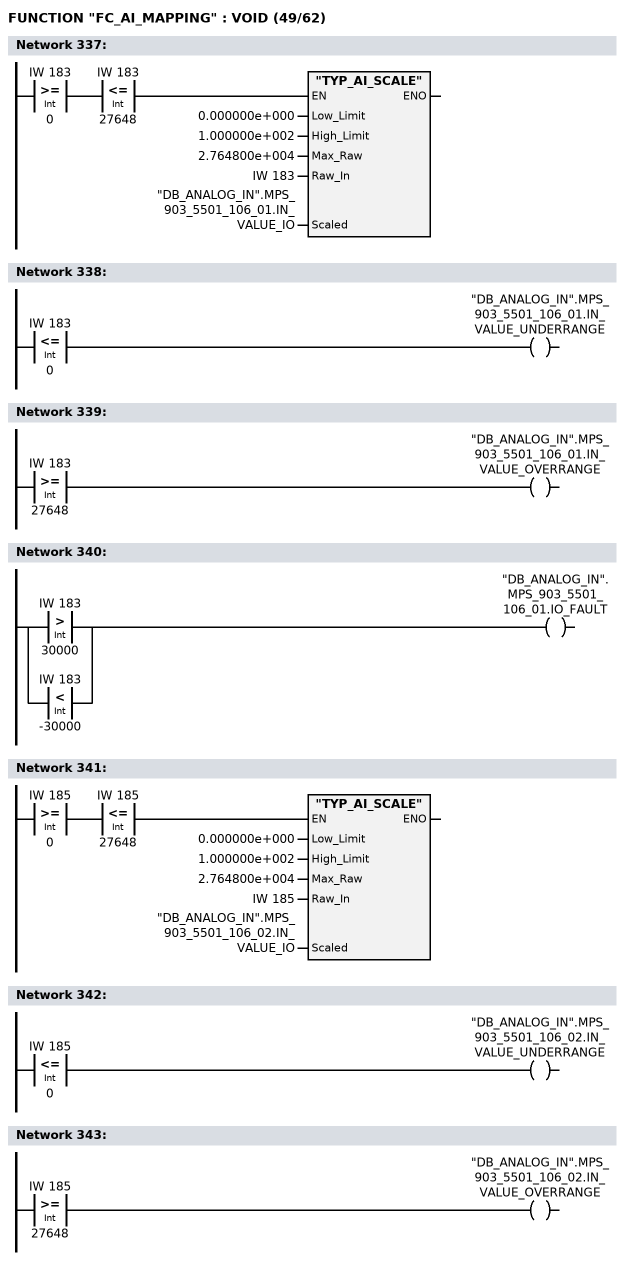

      A(    ;
      L     IW      183;
      L     0;
      >=I   ;
      )     ;
      A(    ;
      L     IW      183;

      L     27648;
      <=I   ;
      )     ;
      JNB   _055;
      CALL "TYP_AI_SCALE" (
           Low_Limit                := 0.000000e+000,
           High_Limit               := 1.000000e+002,
           Max_Raw                  := 2.764800e+004,
           Raw_In                   := IW      183,
           Scaled                   := "DB_ANALOG_IN".MPS_903_5501_106_01.IN_VALUE_IO);
_055: NOP   0;
NETWORK
TITLE =

      L     IW      183;
      L     0;
      <=I   ;
      =     "DB_ANALOG_IN".MPS_903_5501_106_01.IN_VALUE_UNDERRANGE;
NETWORK
TITLE =

      L     IW      183;
      L     27648;
      >=I   ;
      =     "DB_ANALOG_IN".MPS_903_5501_106_01.IN_VALUE_OVERRANGE;
NETWORK
TITLE =

      O(    ;
      L     IW      183;
      L     30000;
      >I    ;
      )     ;
      O(    ;
      L     IW      183;
      L     -30000;
      <I    ;
      )     ;
      =     "DB_ANALOG_IN".MPS_903_5501_106_01.IO_FAULT;

NETWORK
TITLE =

      A(    ;
      L     IW      185;
      L     0;
      >=I   ;
      )     ;
      A(    ;
      L     IW      185;

      L     27648;
      <=I   ;
      )     ;
      JNB   _056;
      CALL "TYP_AI_SCALE" (
           Low_Limit                := 0.000000e+000,
           High_Limit               := 1.000000e+002,
           Max_Raw                  := 2.764800e+004,
           Raw_In                   := IW      185,
           Scaled                   := "DB_ANALOG_IN".MPS_903_5501_106_02.IN_VALUE_IO);
_056: NOP   0;
NETWORK
TITLE =

      L     IW      185;
      L     0;
      <=I   ;
      =     "DB_ANALOG_IN".MPS_903_5501_106_02.IN_VALUE_UNDERRANGE;
NETWORK
TITLE =

      L     IW      185;
      L     27648;
      >=I   ;
      =     "DB_ANALOG_IN".MPS_903_5501_106_02.IN_VALUE_OVERRANGE;
NETWORK
TITLE =
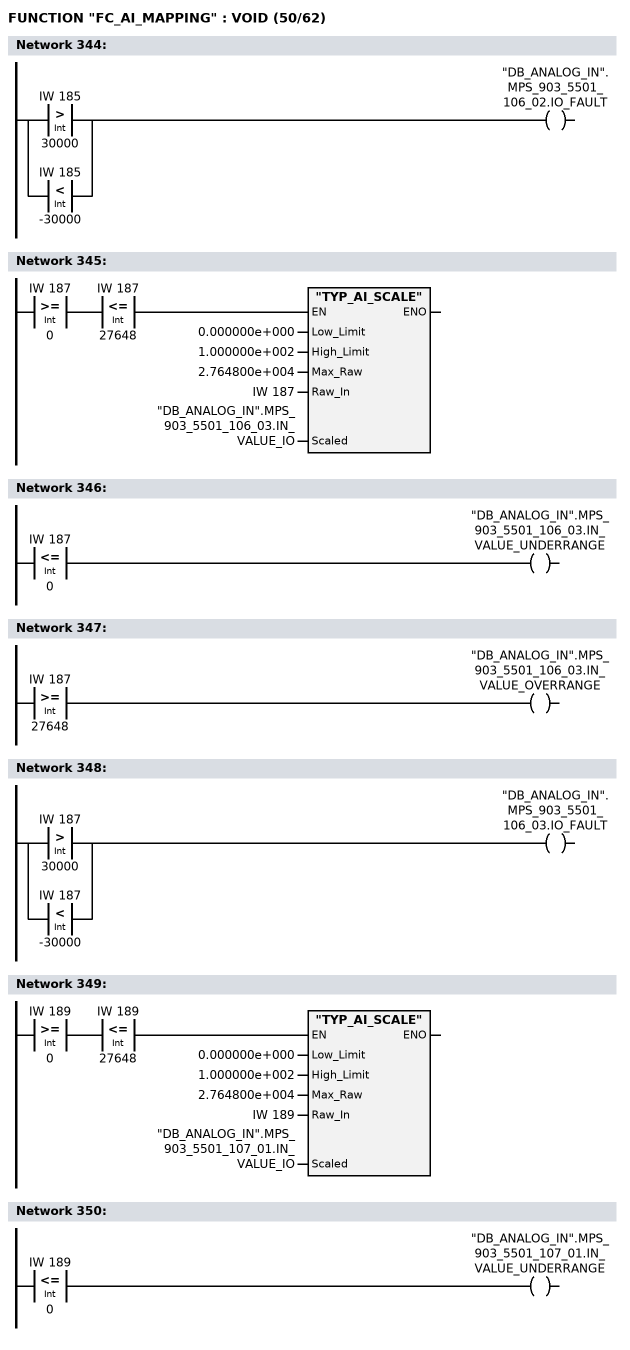

      O(    ;
      L     IW      185;
      L     30000;
      >I    ;
      )     ;
      O(    ;
      L     IW      185;
      L     -30000;
      <I    ;
      )     ;
      =     "DB_ANALOG_IN".MPS_903_5501_106_02.IO_FAULT;

NETWORK
TITLE =

      A(    ;
      L     IW      187;
      L     0;
      >=I   ;
      )     ;
      A(    ;
      L     IW      187;

      L     27648;
      <=I   ;
      )     ;
      JNB   _057;
      CALL "TYP_AI_SCALE" (
           Low_Limit                := 0.000000e+000,
           High_Limit               := 1.000000e+002,
           Max_Raw                  := 2.764800e+004,
           Raw_In                   := IW      187,
           Scaled                   := "DB_ANALOG_IN".MPS_903_5501_106_03.IN_VALUE_IO);
_057: NOP   0;
NETWORK
TITLE =

      L     IW      187;
      L     0;
      <=I   ;
      =     "DB_ANALOG_IN".MPS_903_5501_106_03.IN_VALUE_UNDERRANGE;
NETWORK
TITLE =

      L     IW      187;
      L     27648;
      >=I   ;
      =     "DB_ANALOG_IN".MPS_903_5501_106_03.IN_VALUE_OVERRANGE;
NETWORK
TITLE =

      O(    ;
      L     IW      187;
      L     30000;
      >I    ;
      )     ;
      O(    ;
      L     IW      187;
      L     -30000;
      <I    ;
      )     ;
      =     "DB_ANALOG_IN".MPS_903_5501_106_03.IO_FAULT;

NETWORK
TITLE =

      A(    ;
      L     IW      189;
      L     0;
      >=I   ;
      )     ;
      A(    ;
      L     IW      189;

      L     27648;
      <=I   ;
      )     ;
      JNB   _058;
      CALL "TYP_AI_SCALE" (
           Low_Limit                := 0.000000e+000,
           High_Limit               := 1.000000e+002,
           Max_Raw                  := 2.764800e+004,
           Raw_In                   := IW      189,
           Scaled                   := "DB_ANALOG_IN".MPS_903_5501_107_01.IN_VALUE_IO);
_058: NOP   0;
NETWORK
TITLE =

      L     IW      189;
      L     0;
      <=I   ;
      =     "DB_ANALOG_IN".MPS_903_5501_107_01.IN_VALUE_UNDERRANGE;
NETWORK
TITLE =
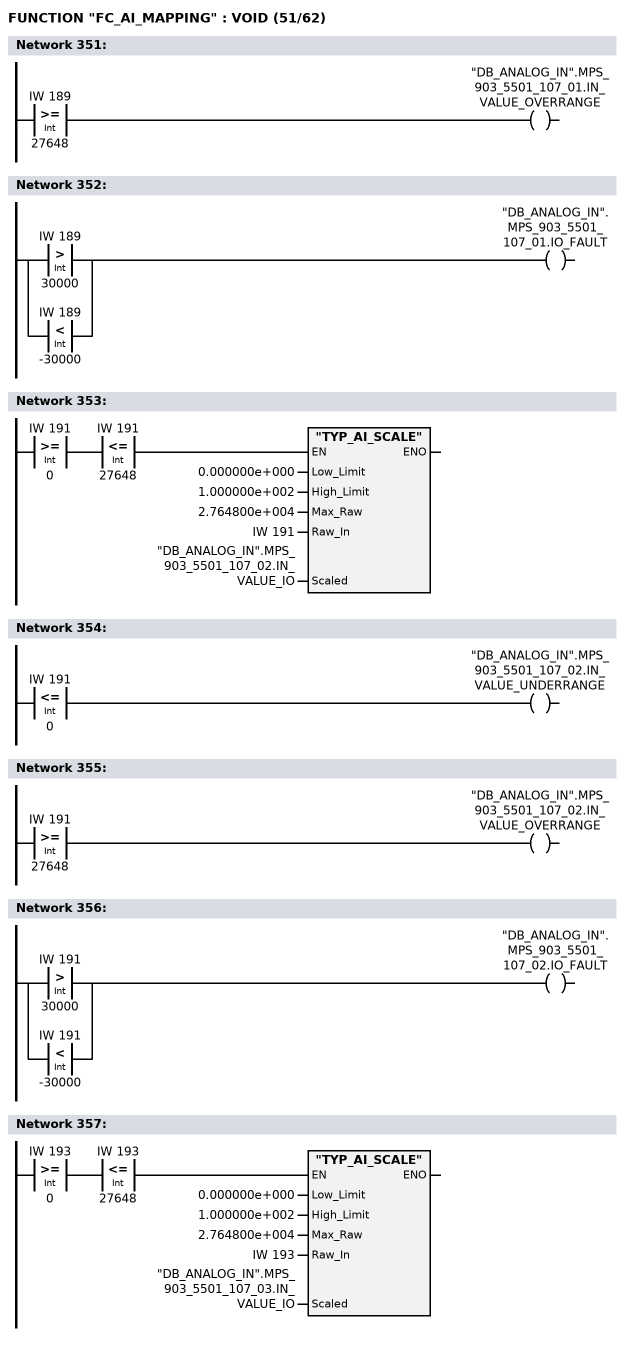

      L     IW      189;
      L     27648;
      >=I   ;
      =     "DB_ANALOG_IN".MPS_903_5501_107_01.IN_VALUE_OVERRANGE;
NETWORK
TITLE =

      O(    ;
      L     IW      189;
      L     30000;
      >I    ;
      )     ;
      O(    ;
      L     IW      189;
      L     -30000;
      <I    ;
      )     ;
      =     "DB_ANALOG_IN".MPS_903_5501_107_01.IO_FAULT;

NETWORK
TITLE =

      A(    ;
      L     IW      191;
      L     0;
      >=I   ;
      )     ;
      A(    ;
      L     IW      191;

      L     27648;
      <=I   ;
      )     ;
      JNB   _059;
      CALL "TYP_AI_SCALE" (
           Low_Limit                := 0.000000e+000,
           High_Limit               := 1.000000e+002,
           Max_Raw                  := 2.764800e+004,
           Raw_In                   := IW      191,
           Scaled                   := "DB_ANALOG_IN".MPS_903_5501_107_02.IN_VALUE_IO);
_059: NOP   0;
NETWORK
TITLE =

      L     IW      191;
      L     0;
      <=I   ;
      =     "DB_ANALOG_IN".MPS_903_5501_107_02.IN_VALUE_UNDERRANGE;
NETWORK
TITLE =

      L     IW      191;
      L     27648;
      >=I   ;
      =     "DB_ANALOG_IN".MPS_903_5501_107_02.IN_VALUE_OVERRANGE;
NETWORK
TITLE =

      O(    ;
      L     IW      191;
      L     30000;
      >I    ;
      )     ;
      O(    ;
      L     IW      191;
      L     -30000;
      <I    ;
      )     ;
      =     "DB_ANALOG_IN".MPS_903_5501_107_02.IO_FAULT;

NETWORK
TITLE =

      A(    ;
      L     IW      193;
      L     0;
      >=I   ;
      )     ;
      A(    ;
      L     IW      193;

      L     27648;
      <=I   ;
      )     ;
      JNB   _05a;
      CALL "TYP_AI_SCALE" (
           Low_Limit                := 0.000000e+000,
           High_Limit               := 1.000000e+002,
           Max_Raw                  := 2.764800e+004,
           Raw_In                   := IW      193,
           Scaled                   := "DB_ANALOG_IN".MPS_903_5501_107_03.IN_VALUE_IO);
_05a: NOP   0;
NETWORK
TITLE =
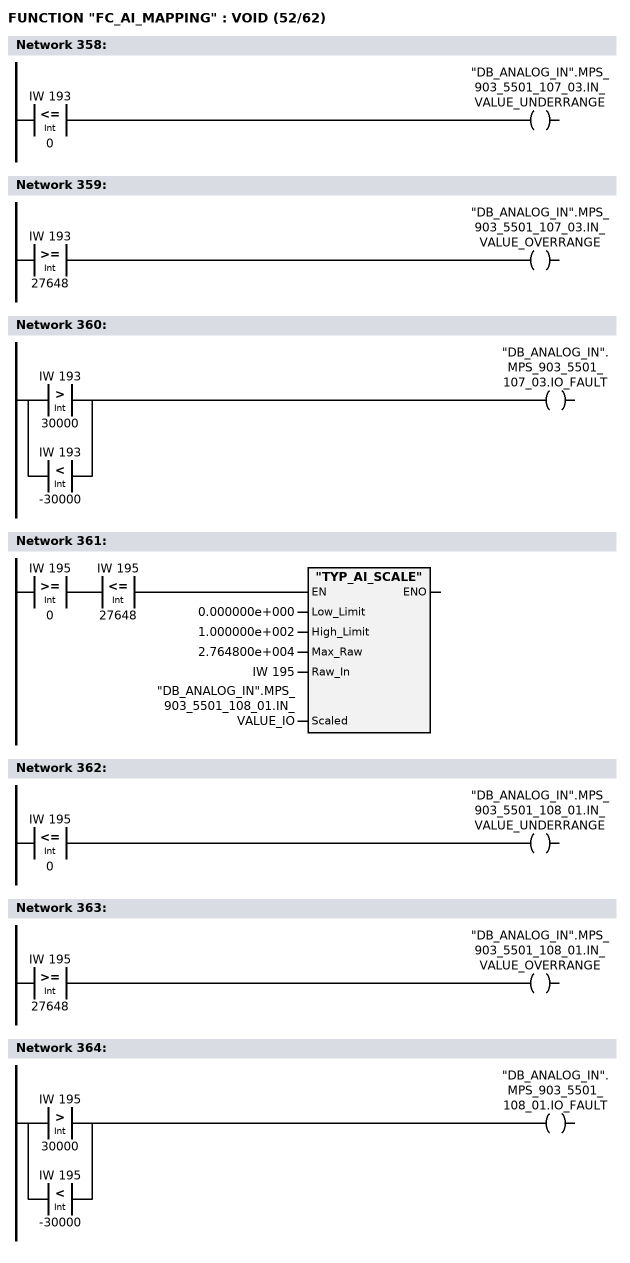

      L     IW      193;
      L     0;
      <=I   ;
      =     "DB_ANALOG_IN".MPS_903_5501_107_03.IN_VALUE_UNDERRANGE;
NETWORK
TITLE =

      L     IW      193;
      L     27648;
      >=I   ;
      =     "DB_ANALOG_IN".MPS_903_5501_107_03.IN_VALUE_OVERRANGE;
NETWORK
TITLE =

      O(    ;
      L     IW      193;
      L     30000;
      >I    ;
      )     ;
      O(    ;
      L     IW      193;
      L     -30000;
      <I    ;
      )     ;
      =     "DB_ANALOG_IN".MPS_903_5501_107_03.IO_FAULT;

NETWORK
TITLE =

      A(    ;
      L     IW      195;
      L     0;
      >=I   ;
      )     ;
      A(    ;
      L     IW      195;

      L     27648;
      <=I   ;
      )     ;
      JNB   _05b;
      CALL "TYP_AI_SCALE" (
           Low_Limit                := 0.000000e+000,
           High_Limit               := 1.000000e+002,
           Max_Raw                  := 2.764800e+004,
           Raw_In                   := IW      195,
           Scaled                   := "DB_ANALOG_IN".MPS_903_5501_108_01.IN_VALUE_IO);
_05b: NOP   0;
NETWORK
TITLE =

      L     IW      195;
      L     0;
      <=I   ;
      =     "DB_ANALOG_IN".MPS_903_5501_108_01.IN_VALUE_UNDERRANGE;
NETWORK
TITLE =

      L     IW      195;
      L     27648;
      >=I   ;
      =     "DB_ANALOG_IN".MPS_903_5501_108_01.IN_VALUE_OVERRANGE;
NETWORK
TITLE =

      O(    ;
      L     IW      195;
      L     30000;
      >I    ;
      )     ;
      O(    ;
      L     IW      195;
      L     -30000;
      <I    ;
      )     ;
      =     "DB_ANALOG_IN".MPS_903_5501_108_01.IO_FAULT;

NETWORK
TITLE =
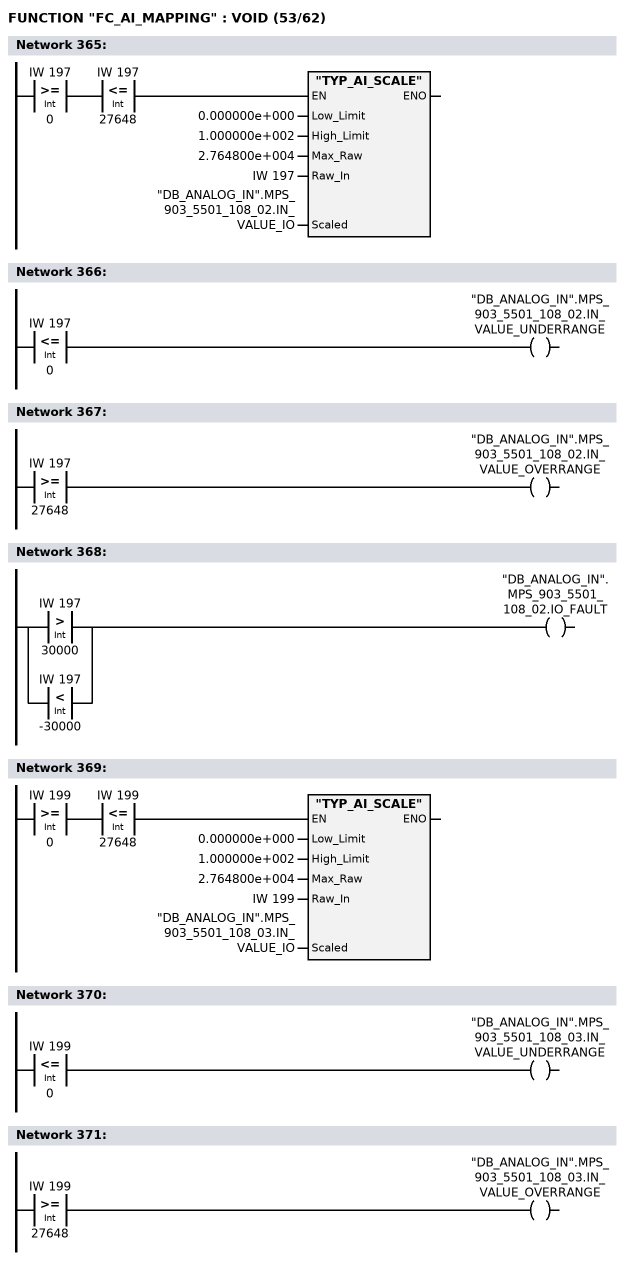

      A(    ;
      L     IW      197;
      L     0;
      >=I   ;
      )     ;
      A(    ;
      L     IW      197;

      L     27648;
      <=I   ;
      )     ;
      JNB   _05c;
      CALL "TYP_AI_SCALE" (
           Low_Limit                := 0.000000e+000,
           High_Limit               := 1.000000e+002,
           Max_Raw                  := 2.764800e+004,
           Raw_In                   := IW      197,
           Scaled                   := "DB_ANALOG_IN".MPS_903_5501_108_02.IN_VALUE_IO);
_05c: NOP   0;
NETWORK
TITLE =

      L     IW      197;
      L     0;
      <=I   ;
      =     "DB_ANALOG_IN".MPS_903_5501_108_02.IN_VALUE_UNDERRANGE;
NETWORK
TITLE =

      L     IW      197;
      L     27648;
      >=I   ;
      =     "DB_ANALOG_IN".MPS_903_5501_108_02.IN_VALUE_OVERRANGE;
NETWORK
TITLE =

      O(    ;
      L     IW      197;
      L     30000;
      >I    ;
      )     ;
      O(    ;
      L     IW      197;
      L     -30000;
      <I    ;
      )     ;
      =     "DB_ANALOG_IN".MPS_903_5501_108_02.IO_FAULT;

NETWORK
TITLE =

      A(    ;
      L     IW      199;
      L     0;
      >=I   ;
      )     ;
      A(    ;
      L     IW      199;

      L     27648;
      <=I   ;
      )     ;
      JNB   _05d;
      CALL "TYP_AI_SCALE" (
           Low_Limit                := 0.000000e+000,
           High_Limit               := 1.000000e+002,
           Max_Raw                  := 2.764800e+004,
           Raw_In                   := IW      199,
           Scaled                   := "DB_ANALOG_IN".MPS_903_5501_108_03.IN_VALUE_IO);
_05d: NOP   0;
NETWORK
TITLE =

      L     IW      199;
      L     0;
      <=I   ;
      =     "DB_ANALOG_IN".MPS_903_5501_108_03.IN_VALUE_UNDERRANGE;
NETWORK
TITLE =

      L     IW      199;
      L     27648;
      >=I   ;
      =     "DB_ANALOG_IN".MPS_903_5501_108_03.IN_VALUE_OVERRANGE;
NETWORK
TITLE =
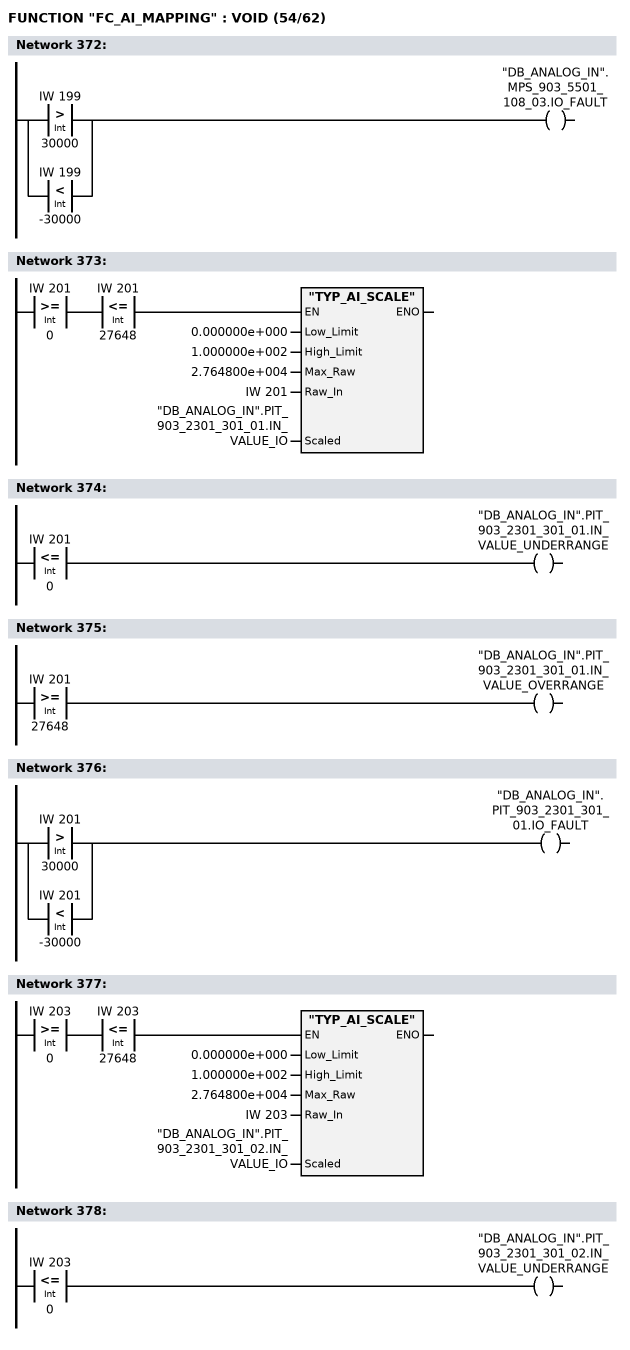

      O(    ;
      L     IW      199;
      L     30000;
      >I    ;
      )     ;
      O(    ;
      L     IW      199;
      L     -30000;
      <I    ;
      )     ;
      =     "DB_ANALOG_IN".MPS_903_5501_108_03.IO_FAULT;

NETWORK
TITLE =

      A(    ;
      L     IW      201;
      L     0;
      >=I   ;
      )     ;
      A(    ;
      L     IW      201;

      L     27648;
      <=I   ;
      )     ;
      JNB   _05e;
      CALL "TYP_AI_SCALE" (
           Low_Limit                := 0.000000e+000,
           High_Limit               := 1.000000e+002,
           Max_Raw                  := 2.764800e+004,
           Raw_In                   := IW      201,
           Scaled                   := "DB_ANALOG_IN".PIT_903_2301_301_01.IN_VALUE_IO);
_05e: NOP   0;
NETWORK
TITLE =

      L     IW      201;
      L     0;
      <=I   ;
      =     "DB_ANALOG_IN".PIT_903_2301_301_01.IN_VALUE_UNDERRANGE;
NETWORK
TITLE =

      L     IW      201;
      L     27648;
      >=I   ;
      =     "DB_ANALOG_IN".PIT_903_2301_301_01.IN_VALUE_OVERRANGE;
NETWORK
TITLE =

      O(    ;
      L     IW      201;
      L     30000;
      >I    ;
      )     ;
      O(    ;
      L     IW      201;
      L     -30000;
      <I    ;
      )     ;
      =     "DB_ANALOG_IN".PIT_903_2301_301_01.IO_FAULT;

NETWORK
TITLE =

      A(    ;
      L     IW      203;
      L     0;
      >=I   ;
      )     ;
      A(    ;
      L     IW      203;

      L     27648;
      <=I   ;
      )     ;
      JNB   _05f;
      CALL "TYP_AI_SCALE" (
           Low_Limit                := 0.000000e+000,
           High_Limit               := 1.000000e+002,
           Max_Raw                  := 2.764800e+004,
           Raw_In                   := IW      203,
           Scaled                   := "DB_ANALOG_IN".PIT_903_2301_301_02.IN_VALUE_IO);
_05f: NOP   0;
NETWORK
TITLE =

      L     IW      203;
      L     0;
      <=I   ;
      =     "DB_ANALOG_IN".PIT_903_2301_301_02.IN_VALUE_UNDERRANGE;
NETWORK
TITLE =
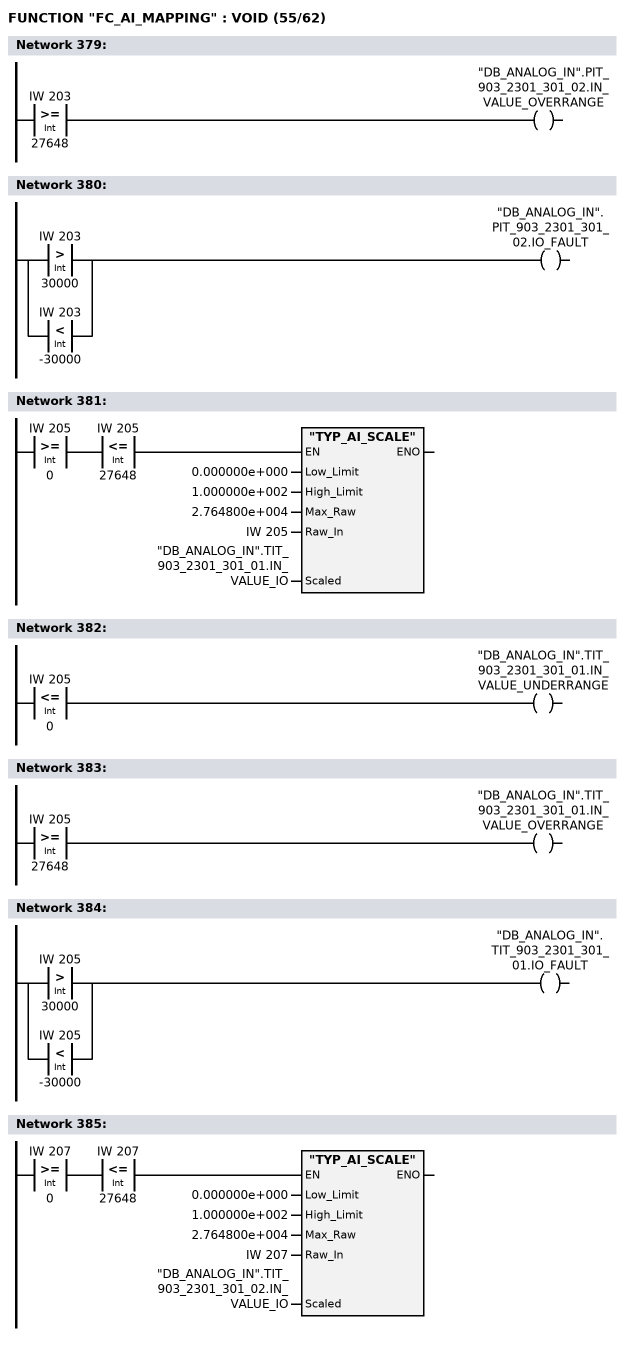

      L     IW      203;
      L     27648;
      >=I   ;
      =     "DB_ANALOG_IN".PIT_903_2301_301_02.IN_VALUE_OVERRANGE;
NETWORK
TITLE =

      O(    ;
      L     IW      203;
      L     30000;
      >I    ;
      )     ;
      O(    ;
      L     IW      203;
      L     -30000;
      <I    ;
      )     ;
      =     "DB_ANALOG_IN".PIT_903_2301_301_02.IO_FAULT;

NETWORK
TITLE =

      A(    ;
      L     IW      205;
      L     0;
      >=I   ;
      )     ;
      A(    ;
      L     IW      205;

      L     27648;
      <=I   ;
      )     ;
      JNB   _060;
      CALL "TYP_AI_SCALE" (
           Low_Limit                := 0.000000e+000,
           High_Limit               := 1.000000e+002,
           Max_Raw                  := 2.764800e+004,
           Raw_In                   := IW      205,
           Scaled                   := "DB_ANALOG_IN".TIT_903_2301_301_01.IN_VALUE_IO);
_060: NOP   0;
NETWORK
TITLE =

      L     IW      205;
      L     0;
      <=I   ;
      =     "DB_ANALOG_IN".TIT_903_2301_301_01.IN_VALUE_UNDERRANGE;
NETWORK
TITLE =

      L     IW      205;
      L     27648;
      >=I   ;
      =     "DB_ANALOG_IN".TIT_903_2301_301_01.IN_VALUE_OVERRANGE;
NETWORK
TITLE =

      O(    ;
      L     IW      205;
      L     30000;
      >I    ;
      )     ;
      O(    ;
      L     IW      205;
      L     -30000;
      <I    ;
      )     ;
      =     "DB_ANALOG_IN".TIT_903_2301_301_01.IO_FAULT;

NETWORK
TITLE =

      A(    ;
      L     IW      207;
      L     0;
      >=I   ;
      )     ;
      A(    ;
      L     IW      207;

      L     27648;
      <=I   ;
      )     ;
      JNB   _061;
      CALL "TYP_AI_SCALE" (
           Low_Limit                := 0.000000e+000,
           High_Limit               := 1.000000e+002,
           Max_Raw                  := 2.764800e+004,
           Raw_In                   := IW      207,
           Scaled                   := "DB_ANALOG_IN".TIT_903_2301_301_02.IN_VALUE_IO);
_061: NOP   0;
NETWORK
TITLE =
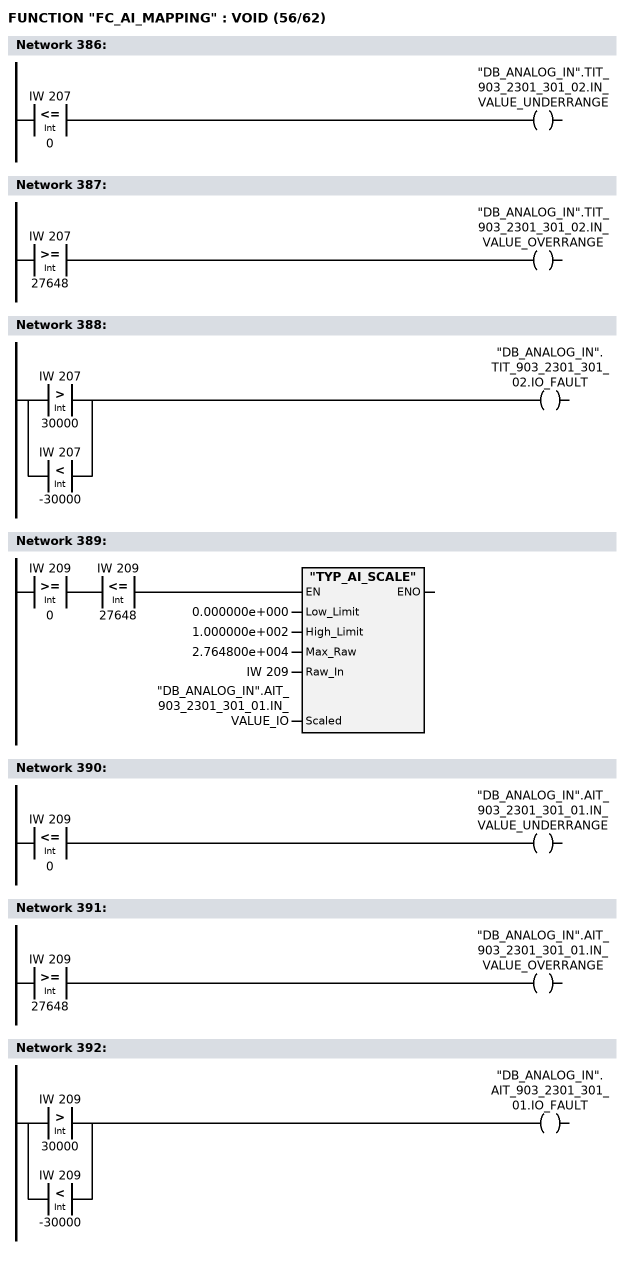

      L     IW      207;
      L     0;
      <=I   ;
      =     "DB_ANALOG_IN".TIT_903_2301_301_02.IN_VALUE_UNDERRANGE;
NETWORK
TITLE =

      L     IW      207;
      L     27648;
      >=I   ;
      =     "DB_ANALOG_IN".TIT_903_2301_301_02.IN_VALUE_OVERRANGE;
NETWORK
TITLE =

      O(    ;
      L     IW      207;
      L     30000;
      >I    ;
      )     ;
      O(    ;
      L     IW      207;
      L     -30000;
      <I    ;
      )     ;
      =     "DB_ANALOG_IN".TIT_903_2301_301_02.IO_FAULT;

NETWORK
TITLE =

      A(    ;
      L     IW      209;
      L     0;
      >=I   ;
      )     ;
      A(    ;
      L     IW      209;

      L     27648;
      <=I   ;
      )     ;
      JNB   _062;
      CALL "TYP_AI_SCALE" (
           Low_Limit                := 0.000000e+000,
           High_Limit               := 1.000000e+002,
           Max_Raw                  := 2.764800e+004,
           Raw_In                   := IW      209,
           Scaled                   := "DB_ANALOG_IN".AIT_903_2301_301_01.IN_VALUE_IO);
_062: NOP   0;
NETWORK
TITLE =

      L     IW      209;
      L     0;
      <=I   ;
      =     "DB_ANALOG_IN".AIT_903_2301_301_01.IN_VALUE_UNDERRANGE;
NETWORK
TITLE =

      L     IW      209;
      L     27648;
      >=I   ;
      =     "DB_ANALOG_IN".AIT_903_2301_301_01.IN_VALUE_OVERRANGE;
NETWORK
TITLE =

      O(    ;
      L     IW      209;
      L     30000;
      >I    ;
      )     ;
      O(    ;
      L     IW      209;
      L     -30000;
      <I    ;
      )     ;
      =     "DB_ANALOG_IN".AIT_903_2301_301_01.IO_FAULT;

NETWORK
TITLE =
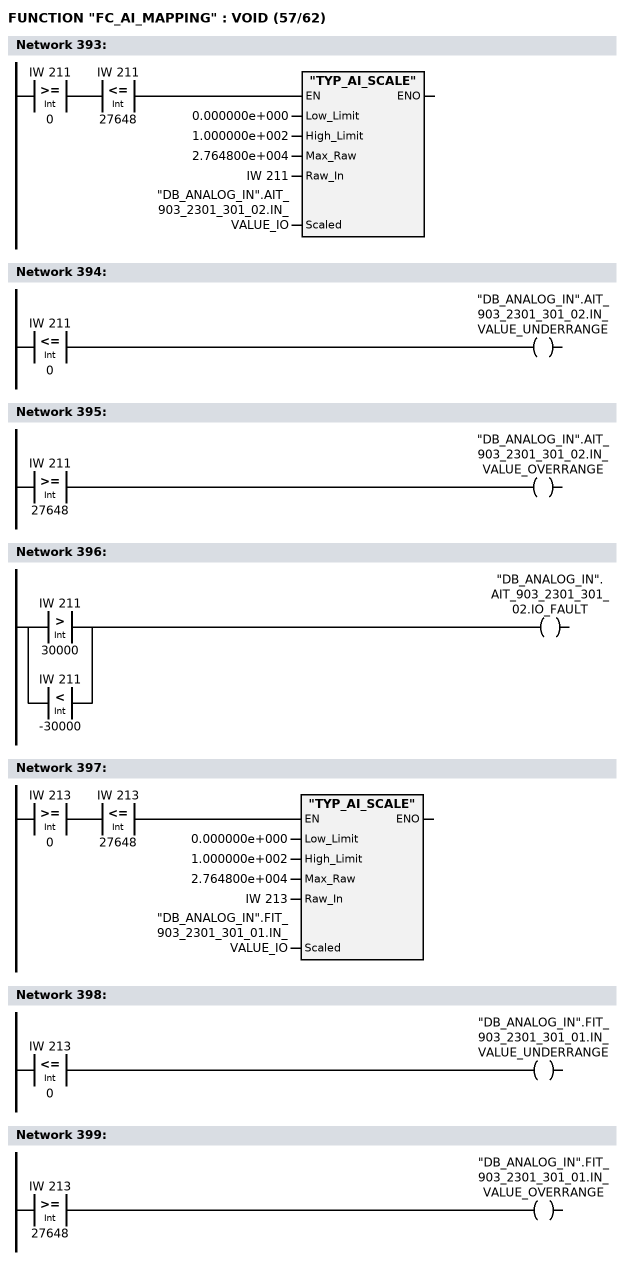

      A(    ;
      L     IW      211;
      L     0;
      >=I   ;
      )     ;
      A(    ;
      L     IW      211;

      L     27648;
      <=I   ;
      )     ;
      JNB   _063;
      CALL "TYP_AI_SCALE" (
           Low_Limit                := 0.000000e+000,
           High_Limit               := 1.000000e+002,
           Max_Raw                  := 2.764800e+004,
           Raw_In                   := IW      211,
           Scaled                   := "DB_ANALOG_IN".AIT_903_2301_301_02.IN_VALUE_IO);
_063: NOP   0;
NETWORK
TITLE =

      L     IW      211;
      L     0;
      <=I   ;
      =     "DB_ANALOG_IN".AIT_903_2301_301_02.IN_VALUE_UNDERRANGE;
NETWORK
TITLE =

      L     IW      211;
      L     27648;
      >=I   ;
      =     "DB_ANALOG_IN".AIT_903_2301_301_02.IN_VALUE_OVERRANGE;
NETWORK
TITLE =

      O(    ;
      L     IW      211;
      L     30000;
      >I    ;
      )     ;
      O(    ;
      L     IW      211;
      L     -30000;
      <I    ;
      )     ;
      =     "DB_ANALOG_IN".AIT_903_2301_301_02.IO_FAULT;

NETWORK
TITLE =

      A(    ;
      L     IW      213;
      L     0;
      >=I   ;
      )     ;
      A(    ;
      L     IW      213;

      L     27648;
      <=I   ;
      )     ;
      JNB   _064;
      CALL "TYP_AI_SCALE" (
           Low_Limit                := 0.000000e+000,
           High_Limit               := 1.000000e+002,
           Max_Raw                  := 2.764800e+004,
           Raw_In                   := IW      213,
           Scaled                   := "DB_ANALOG_IN".FIT_903_2301_301_01.IN_VALUE_IO);
_064: NOP   0;
NETWORK
TITLE =

      L     IW      213;
      L     0;
      <=I   ;
      =     "DB_ANALOG_IN".FIT_903_2301_301_01.IN_VALUE_UNDERRANGE;
NETWORK
TITLE =

      L     IW      213;
      L     27648;
      >=I   ;
      =     "DB_ANALOG_IN".FIT_903_2301_301_01.IN_VALUE_OVERRANGE;
NETWORK
TITLE =
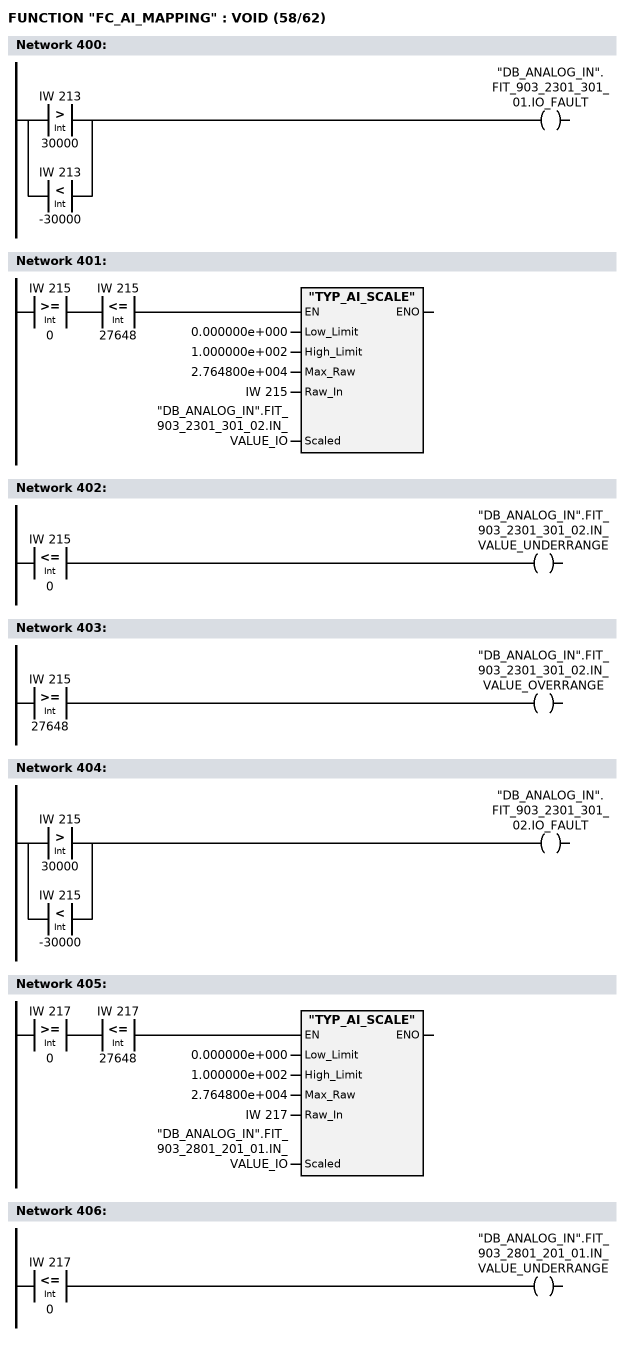

      O(    ;
      L     IW      213;
      L     30000;
      >I    ;
      )     ;
      O(    ;
      L     IW      213;
      L     -30000;
      <I    ;
      )     ;
      =     "DB_ANALOG_IN".FIT_903_2301_301_01.IO_FAULT;

NETWORK
TITLE =

      A(    ;
      L     IW      215;
      L     0;
      >=I   ;
      )     ;
      A(    ;
      L     IW      215;

      L     27648;
      <=I   ;
      )     ;
      JNB   _065;
      CALL "TYP_AI_SCALE" (
           Low_Limit                := 0.000000e+000,
           High_Limit               := 1.000000e+002,
           Max_Raw                  := 2.764800e+004,
           Raw_In                   := IW      215,
           Scaled                   := "DB_ANALOG_IN".FIT_903_2301_301_02.IN_VALUE_IO);
_065: NOP   0;
NETWORK
TITLE =

      L     IW      215;
      L     0;
      <=I   ;
      =     "DB_ANALOG_IN".FIT_903_2301_301_02.IN_VALUE_UNDERRANGE;
NETWORK
TITLE =

      L     IW      215;
      L     27648;
      >=I   ;
      =     "DB_ANALOG_IN".FIT_903_2301_301_02.IN_VALUE_OVERRANGE;
NETWORK
TITLE =

      O(    ;
      L     IW      215;
      L     30000;
      >I    ;
      )     ;
      O(    ;
      L     IW      215;
      L     -30000;
      <I    ;
      )     ;
      =     "DB_ANALOG_IN".FIT_903_2301_301_02.IO_FAULT;

NETWORK
TITLE =

      A(    ;
      L     IW      217;
      L     0;
      >=I   ;
      )     ;
      A(    ;
      L     IW      217;

      L     27648;
      <=I   ;
      )     ;
      JNB   _066;
      CALL "TYP_AI_SCALE" (
           Low_Limit                := 0.000000e+000,
           High_Limit               := 1.000000e+002,
           Max_Raw                  := 2.764800e+004,
           Raw_In                   := IW      217,
           Scaled                   := "DB_ANALOG_IN".FIT_903_2801_201_01.IN_VALUE_IO);
_066: NOP   0;
NETWORK
TITLE =

      L     IW      217;
      L     0;
      <=I   ;
      =     "DB_ANALOG_IN".FIT_903_2801_201_01.IN_VALUE_UNDERRANGE;
NETWORK
TITLE =
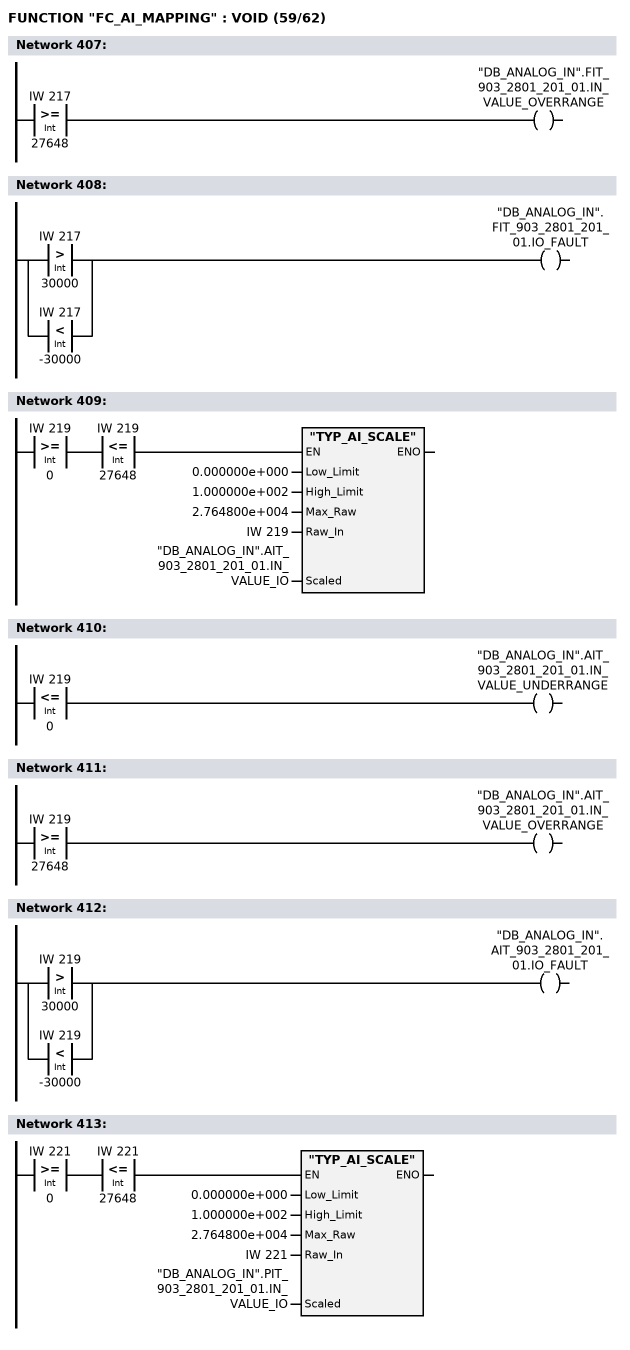

      L     IW      217;
      L     27648;
      >=I   ;
      =     "DB_ANALOG_IN".FIT_903_2801_201_01.IN_VALUE_OVERRANGE;
NETWORK
TITLE =

      O(    ;
      L     IW      217;
      L     30000;
      >I    ;
      )     ;
      O(    ;
      L     IW      217;
      L     -30000;
      <I    ;
      )     ;
      =     "DB_ANALOG_IN".FIT_903_2801_201_01.IO_FAULT;

NETWORK
TITLE =

      A(    ;
      L     IW      219;
      L     0;
      >=I   ;
      )     ;
      A(    ;
      L     IW      219;

      L     27648;
      <=I   ;
      )     ;
      JNB   _067;
      CALL "TYP_AI_SCALE" (
           Low_Limit                := 0.000000e+000,
           High_Limit               := 1.000000e+002,
           Max_Raw                  := 2.764800e+004,
           Raw_In                   := IW      219,
           Scaled                   := "DB_ANALOG_IN".AIT_903_2801_201_01.IN_VALUE_IO);
_067: NOP   0;
NETWORK
TITLE =

      L     IW      219;
      L     0;
      <=I   ;
      =     "DB_ANALOG_IN".AIT_903_2801_201_01.IN_VALUE_UNDERRANGE;
NETWORK
TITLE =

      L     IW      219;
      L     27648;
      >=I   ;
      =     "DB_ANALOG_IN".AIT_903_2801_201_01.IN_VALUE_OVERRANGE;
NETWORK
TITLE =

      O(    ;
      L     IW      219;
      L     30000;
      >I    ;
      )     ;
      O(    ;
      L     IW      219;
      L     -30000;
      <I    ;
      )     ;
      =     "DB_ANALOG_IN".AIT_903_2801_201_01.IO_FAULT;

NETWORK
TITLE =

      A(    ;
      L     IW      221;
      L     0;
      >=I   ;
      )     ;
      A(    ;
      L     IW      221;

      L     27648;
      <=I   ;
      )     ;
      JNB   _068;
      CALL "TYP_AI_SCALE" (
           Low_Limit                := 0.000000e+000,
           High_Limit               := 1.000000e+002,
           Max_Raw                  := 2.764800e+004,
           Raw_In                   := IW      221,
           Scaled                   := "DB_ANALOG_IN".PIT_903_2801_201_01.IN_VALUE_IO);
_068: NOP   0;
NETWORK
TITLE =
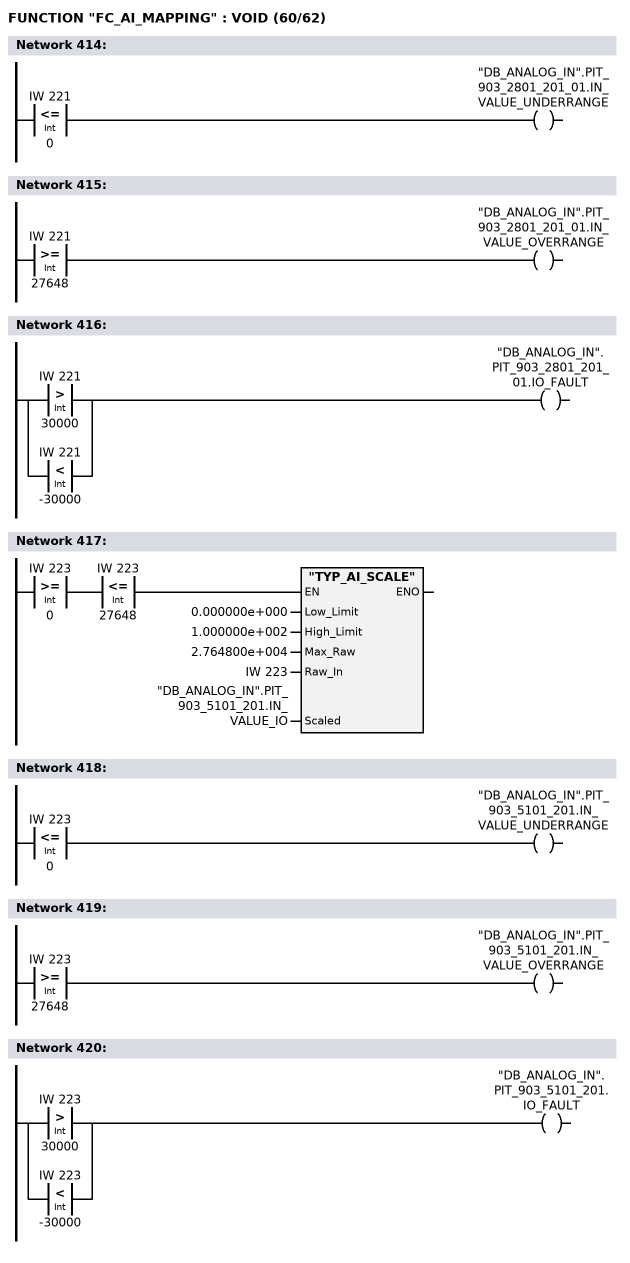

      L     IW      221;
      L     0;
      <=I   ;
      =     "DB_ANALOG_IN".PIT_903_2801_201_01.IN_VALUE_UNDERRANGE;
NETWORK
TITLE =

      L     IW      221;
      L     27648;
      >=I   ;
      =     "DB_ANALOG_IN".PIT_903_2801_201_01.IN_VALUE_OVERRANGE;
NETWORK
TITLE =

      O(    ;
      L     IW      221;
      L     30000;
      >I    ;
      )     ;
      O(    ;
      L     IW      221;
      L     -30000;
      <I    ;
      )     ;
      =     "DB_ANALOG_IN".PIT_903_2801_201_01.IO_FAULT;

NETWORK
TITLE =

      A(    ;
      L     IW      223;
      L     0;
      >=I   ;
      )     ;
      A(    ;
      L     IW      223;

      L     27648;
      <=I   ;
      )     ;
      JNB   _069;
      CALL "TYP_AI_SCALE" (
           Low_Limit                := 0.000000e+000,
           High_Limit               := 1.000000e+002,
           Max_Raw                  := 2.764800e+004,
           Raw_In                   := IW      223,
           Scaled                   := "DB_ANALOG_IN".PIT_903_5101_201.IN_VALUE_IO);
_069: NOP   0;
NETWORK
TITLE =

      L     IW      223;
      L     0;
      <=I   ;
      =     "DB_ANALOG_IN".PIT_903_5101_201.IN_VALUE_UNDERRANGE;
NETWORK
TITLE =

      L     IW      223;
      L     27648;
      >=I   ;
      =     "DB_ANALOG_IN".PIT_903_5101_201.IN_VALUE_OVERRANGE;
NETWORK
TITLE =

      O(    ;
      L     IW      223;
      L     30000;
      >I    ;
      )     ;
      O(    ;
      L     IW      223;
      L     -30000;
      <I    ;
      )     ;
      =     "DB_ANALOG_IN".PIT_903_5101_201.IO_FAULT;

NETWORK
TITLE =
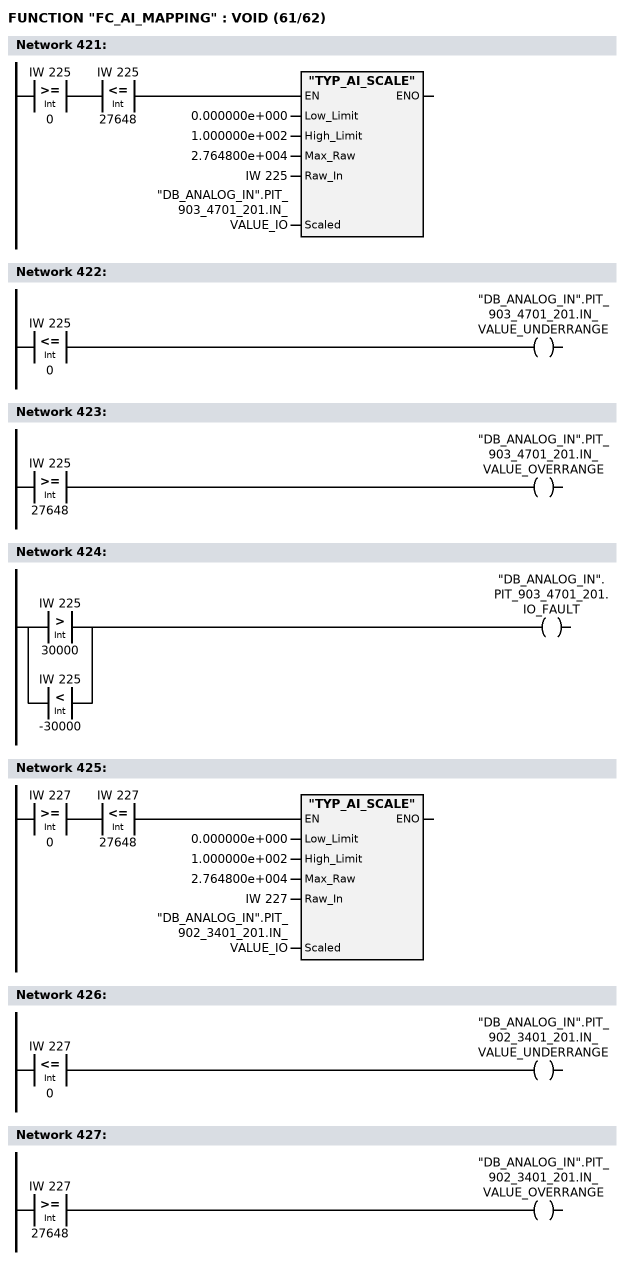

      A(    ;
      L     IW      225;
      L     0;
      >=I   ;
      )     ;
      A(    ;
      L     IW      225;

      L     27648;
      <=I   ;
      )     ;
      JNB   _06a;
      CALL "TYP_AI_SCALE" (
           Low_Limit                := 0.000000e+000,
           High_Limit               := 1.000000e+002,
           Max_Raw                  := 2.764800e+004,
           Raw_In                   := IW      225,
           Scaled                   := "DB_ANALOG_IN".PIT_903_4701_201.IN_VALUE_IO);
_06a: NOP   0;
NETWORK
TITLE =

      L     IW      225;
      L     0;
      <=I   ;
      =     "DB_ANALOG_IN".PIT_903_4701_201.IN_VALUE_UNDERRANGE;
NETWORK
TITLE =

      L     IW      225;
      L     27648;
      >=I   ;
      =     "DB_ANALOG_IN".PIT_903_4701_201.IN_VALUE_OVERRANGE;
NETWORK
TITLE =

      O(    ;
      L     IW      225;
      L     30000;
      >I    ;
      )     ;
      O(    ;
      L     IW      225;
      L     -30000;
      <I    ;
      )     ;
      =     "DB_ANALOG_IN".PIT_903_4701_201.IO_FAULT;

NETWORK
TITLE =

      A(    ;
      L     IW      227;
      L     0;
      >=I   ;
      )     ;
      A(    ;
      L     IW      227;

      L     27648;
      <=I   ;
      )     ;
      JNB   _06b;
      CALL "TYP_AI_SCALE" (
           Low_Limit                := 0.000000e+000,
           High_Limit               := 1.000000e+002,
           Max_Raw                  := 2.764800e+004,
           Raw_In                   := IW      227,
           Scaled                   := "DB_ANALOG_IN".PIT_902_3401_201.IN_VALUE_IO);
_06b: NOP   0;
NETWORK
TITLE =

      L     IW      227;
      L     0;
      <=I   ;
      =     "DB_ANALOG_IN".PIT_902_3401_201.IN_VALUE_UNDERRANGE;
NETWORK
TITLE =

      L     IW      227;
      L     27648;
      >=I   ;
      =     "DB_ANALOG_IN".PIT_902_3401_201.IN_VALUE_OVERRANGE;
NETWORK
TITLE =
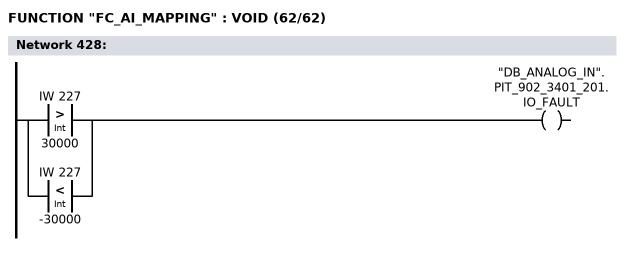

      O(    ;
      L     IW      227;
      L     30000;
      >I    ;
      )     ;
      O(    ;
      L     IW      227;
      L     -30000;
      <I    ;
      )     ;
      =     "DB_ANALOG_IN".PIT_902_3401_201.IO_FAULT;
END_FUNCTION
